// TIA Portal V19 export
FUNCTION_BLOCK "A0302_Centratori_FB"   // FB92, LAD
TITLE = <<< GESTIONE CENTRATORI >>>
// stored: MemoryReserve 100, SetENOAutomatically false
   VAR_INPUT
      AreaInterface : "AreaInterface";
      ZSI : "udt_ZoneSafetyInterface";
      DSI : "udt_DeviceSafetyInterface";
      DataIn : Struct
         OP : "OP_PB";
      END_STRUCT;
      CIn : Struct
         Manager : Struct
            Sollevamento : "ValveMachine_Manager";
            Centraggio : "ValveMachine_Manager";
         END_STRUCT;
         SemiAut_Pb : Bool;
         Rulliera : Struct
            Coda : Struct
               Sens : Struct
                  FTC_Rall : Bool;   // Sensori presenza materiale banco rallentamento ingresso
                  FTC_Prox_Ing : Bool;   // Sensori presenza materiale banco limite ingresso
               END_STRUCT;
            END_STRUCT;
            Centro : Struct
               Sens : Struct
                  FTC_Centrale : Bool;   // 2010BF1 - I50.2
               END_STRUCT;
            END_STRUCT;
         END_STRUCT;
         CarroPareggCoda : Struct
            Ax : "Positioning_DOL_Machine_COut";
            Bloccaggio : "ValveMachine_COut";
            BattutaVerticale : "ValveMachine_COut";
            PareggiatoreLong : "ValveMachine_COut";
            Sens : Struct
               FTC_Ingombro_In : Bool;   // 2012BF1 - I50.0
               FTC_Ingombro_Out : Bool;   // 2012BF2 - I50.1
               PresenzaMat : Bool;   // FC presenza materiale agganciato lato paregg coda
            END_STRUCT;
         END_STRUCT;
         CarroPareggTesta : Struct
            Ax : "Positioning_DOL_Machine_COut";
            Bloccaggio : "ValveMachine_COut";
            Centraggio : "ValveMachine_COut";
            Sollevatore : "ValveMachine_COut";
            Sens : Struct
               FTC1_Rall : Bool;   // 2010BF2 - I50.3
               FTC2_Prox_Ls : Bool;   // 2010BF3 - I50.4
               PresenzaMat : Bool;   // FC presenza materiale agganciato lato paregg testa
            END_STRUCT;
         END_STRUCT;
         BTrk : Struct
            ZoneA0302Entry_Empty : Bool;
            ZoneA0302Exit_Empty : Bool;
         END_STRUCT;
      END_STRUCT;
      Config : Struct
         Centraggio : Array[1..3] of "ValveMachine_Config";
         Sollevamento : Array[1..3] of "ValveMachine_Config";
         DelayMissingCondition : Time;
         WorkWindows : Struct   // Finestre di disattivazione Centratore 1 e 3 in funzione dei Carri
            Coda : Struct
               Min : LReal;
               Max : LReal;
            END_STRUCT;
            Testa : Struct
               Min : LReal;
               Max : LReal;
            END_STRUCT;
         END_STRUCT;
      END_STRUCT;
   END_VAR
   VAR_OUTPUT
      MachineInterface : "MachineInterface";
      COut : Struct
         Centratori : "ValveMachine_COut";
         Centraggio : "ValveMachine_COut";
         Sollevamento : "ValveMachine_COut";
      END_STRUCT;
   END_VAR
   VAR
      Alarm : Struct
         Centraggio : Array[1..3] of "ValveAlr";
         Sollevamento : Array[1..3] of "ValveAlr";
      END_STRUCT;
      Warning : Struct
         Centratore : Array[1..3] of "ValveMachine_Wng";
         Sollevamento : Array[1..3] of "ValveMachine_Wng";
         OP_REST_Centr_MissingCnd : Bool;   // Mancanza comando arresto
         OP_WORK_Centr_MissingCnd : Bool;   // Mancanza consenso lavoro
         OP_REST_Sollev_MissingCnd : Bool;   // Mancanza comando arresto
         OP_WORK_Sollev_MissingCnd : Bool;   // Mancanza consenso lavoro
      END_STRUCT;
      HMI : Struct
         Selection : Struct   // 0=Disable / 1=Enable Pin
            Centraggio : Array[1..3] of Bool;
            Sollevamento : Array[1..3] of Bool;
         END_STRUCT;
         Centratori_Sts : "UDT_HMI-Sts_ValvePosA0301";
         Centraggio_Sts { S7_SetPoint := 'True'} : "UDT_HMI-Sts_ValvePosA0301";
         Sollevamento_Sts { S7_SetPoint := 'True'} : "UDT_HMI-Sts_ValvePosA0301";
      END_STRUCT;
      Centraggio : Array[1..3] of "ValveMachine_FB";
      Sollevamento { S7_SetPoint := 'True'} : Array[1..3] of "ValveMachine_FB";
      Sts : Struct
         Centraggio : Struct
            OP_Rest_Cnd : Bool;
            Op_Work_Cnd : Bool;
         END_STRUCT;
         Sollevamento : Struct
            OP_Rest_Cnd : Bool;
            Op_Work_Cnd : Bool;
         END_STRUCT;
         Centratori_Alarm : Bool;
         Centraggio_AlarmPresence : Bool;
         Sollevamento_AlarmPresence : Bool;
         OP_CanMoveFreely : Bool;
      END_STRUCT;
      Ctrl : Struct
         Centraggio : Struct
            OP_Rest_Man : Bool;
            OP_Work_Man : Bool;
            OP_Rest_Aut : Bool;
            OP_Work_Aut : Bool;
            OP_Rest : Bool;
            OP_Work : Bool;
         END_STRUCT;
         Sollevamento : Struct
            OP_Rest_Man : Bool;
            OP_Work_Man : Bool;
            OP_Rest_Aut : Bool;
            OP_Work_Aut : Bool;
            OP_Rest : Bool;
            OP_Work : Bool;
         END_STRUCT;
      END_STRUCT;
      AUX : Struct
         Centraggio : Struct
            OP_Rest_PB : Bool;
            OP_Work_PB : Bool;
         END_STRUCT;
         Sollevamento : Struct
            OP_Rest_PB : Bool;
            OP_Work_PB : Bool;
         END_STRUCT;
      END_STRUCT;
      TON_OP_REST_Centr_MissingCnd { S7_SetPoint := 'True'} : TON_TIME;
      TON_OP_WORK_Centr_MissingCnd { S7_SetPoint := 'True'} : TON_TIME;
      TON_OP_REST_Sollev_MissingCnd { S7_SetPoint := 'True'} : TON_TIME;
      TON_OP_WORK_Sollev_MissingCnd { S7_SetPoint := 'True'} : TON_TIME;
      DelayMissingCondition : Time;
      TON_Anticipi : Struct
         Work : Struct
            Sollevamento : Array[1..3] of IEC_TIMER;
            Centraggio : Array[1..3] of IEC_TIMER;
         END_STRUCT;
         Rest : Struct
            Sollevamento : Array[1..3] of IEC_TIMER;
            Centraggio : Array[1..3] of IEC_TIMER;
         END_STRUCT;
      END_STRUCT;
   END_VAR
   VAR_TEMP
      PE : Struct
         Centraggio : Struct
            OP_Rest_PB : Bool;
            OP_Work_PB : Bool;
         END_STRUCT;
         Sollevamento : Struct
            OP_Rest_PB : Bool;
            OP_Work_PB : Bool;
         END_STRUCT;
      END_STRUCT;
   END_VAR
   // // Centraggio[1] : Centraggio 1 Coda
   // // Centraggio[2] : Centraggio 2 Centrale
   // // Centraggio[3] : Centraggio 3 Testa
   VAR_TEMP   // added for the SCL form of the ladder/FBD networks
      _w1 : Bool;
      _w2 : Bool;
      _w3 : Bool;
   END_VAR
BEGIN

REGION Network 1: Anticipi Movimento LAVORO
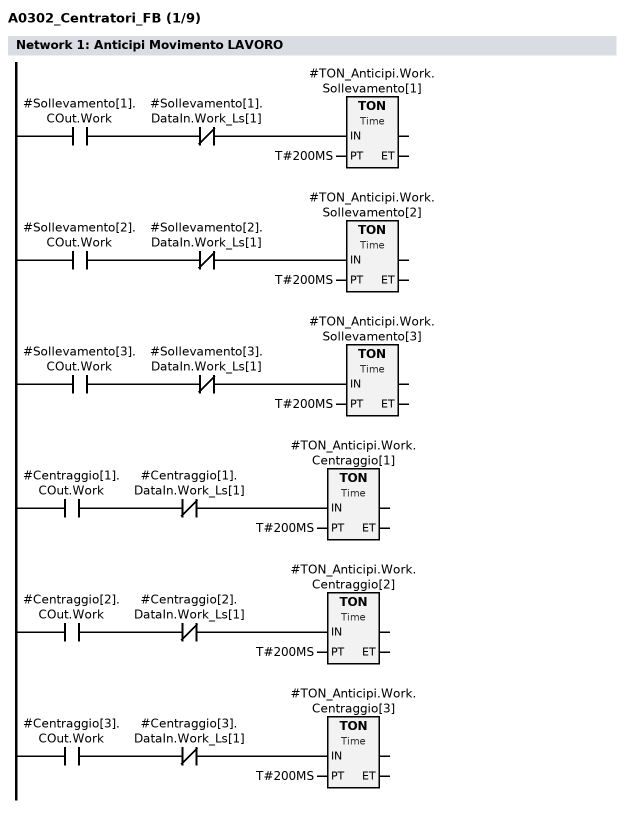
   RUNG wire#powerrail
      Contact( #Sollevamento[1].COut.Work )
      I_Contact( #Sollevamento[1].DataIn.Work_Ls[1] )
      { S7_Templates := "time_type := Time" } #TON_Anticipi.Work.Sollevamento[1].TON(pt := T#200MS, et =>)
   END_RUNG
   RUNG wire#powerrail
      Contact( #Sollevamento[2].COut.Work )
      I_Contact( #Sollevamento[2].DataIn.Work_Ls[1] )
      { S7_Templates := "time_type := Time" } #TON_Anticipi.Work.Sollevamento[2].TON(pt := T#200MS, et =>)
   END_RUNG
   RUNG wire#powerrail
      Contact( #Sollevamento[3].COut.Work )
      I_Contact( #Sollevamento[3].DataIn.Work_Ls[1] )
      { S7_Templates := "time_type := Time" } #TON_Anticipi.Work.Sollevamento[3].TON(pt := T#200MS, et =>)
   END_RUNG
   RUNG wire#powerrail
      Contact( #Centraggio[1].COut.Work )
      I_Contact( #Centraggio[1].DataIn.Work_Ls[1] )
      { S7_Templates := "time_type := Time" } #TON_Anticipi.Work.Centraggio[1].TON(pt := T#200MS, et =>)
   END_RUNG
   RUNG wire#powerrail
      Contact( #Centraggio[2].COut.Work )
      I_Contact( #Centraggio[2].DataIn.Work_Ls[1] )
      { S7_Templates := "time_type := Time" } #TON_Anticipi.Work.Centraggio[2].TON(pt := T#200MS, et =>)
   END_RUNG
   RUNG wire#powerrail
      Contact( #Centraggio[3].COut.Work )
      I_Contact( #Centraggio[3].DataIn.Work_Ls[1] )
      { S7_Templates := "time_type := Time" } #TON_Anticipi.Work.Centraggio[3].TON(pt := T#200MS, et =>)
   END_RUNG
   // the same network as SCL:
   #TON_Anticipi.Work.Sollevamento[1].TON(IN := #Sollevamento[1].COut.Work AND NOT #Sollevamento[1].DataIn.Work_Ls[1],
                           PT := T#200MS);
   #TON_Anticipi.Work.Sollevamento[2].TON(IN := #Sollevamento[2].COut.Work AND NOT #Sollevamento[2].DataIn.Work_Ls[1],
                           PT := T#200MS);
   #TON_Anticipi.Work.Sollevamento[3].TON(IN := #Sollevamento[3].COut.Work AND NOT #Sollevamento[3].DataIn.Work_Ls[1],
                           PT := T#200MS);
   #TON_Anticipi.Work.Centraggio[1].TON(IN := #Centraggio[1].COut.Work AND NOT #Centraggio[1].DataIn.Work_Ls[1],
                           PT := T#200MS);
   #TON_Anticipi.Work.Centraggio[2].TON(IN := #Centraggio[2].COut.Work AND NOT #Centraggio[2].DataIn.Work_Ls[1],
                           PT := T#200MS);
   #TON_Anticipi.Work.Centraggio[3].TON(IN := #Centraggio[3].COut.Work AND NOT #Centraggio[3].DataIn.Work_Ls[1],
                           PT := T#200MS);
END_REGION

REGION Network 2: Anticipi Movimento RIPOSO
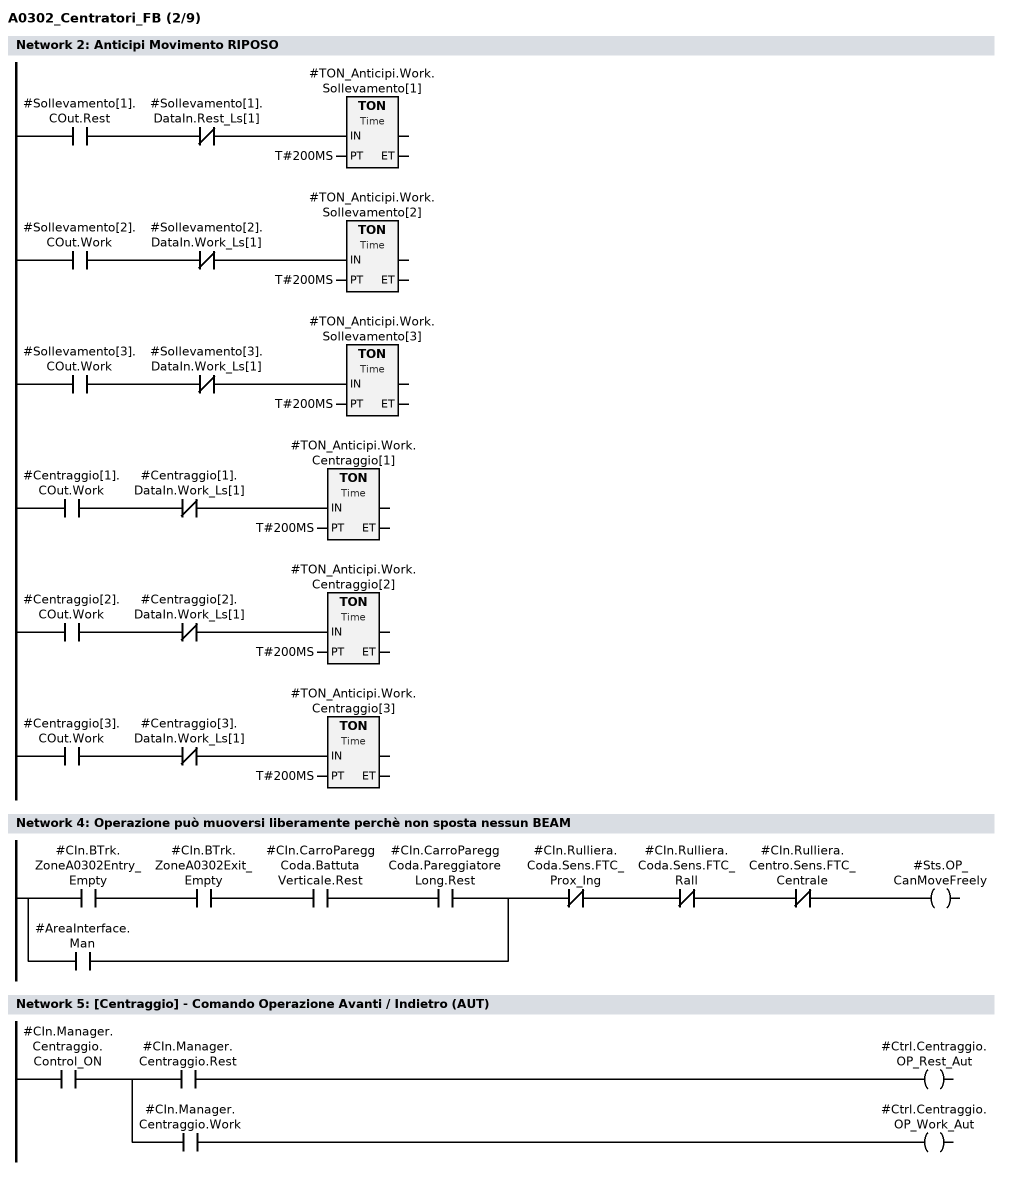
   RUNG wire#powerrail
      Contact( #Sollevamento[1].COut.Rest )
      I_Contact( #Sollevamento[1].DataIn.Rest_Ls[1] )
      { S7_Templates := "time_type := Time" } #TON_Anticipi.Work.Sollevamento[1].TON(pt := T#200MS, et =>)
   END_RUNG
   RUNG wire#powerrail
      Contact( #Sollevamento[2].COut.Work )
      I_Contact( #Sollevamento[2].DataIn.Work_Ls[1] )
      { S7_Templates := "time_type := Time" } #TON_Anticipi.Work.Sollevamento[2].TON(pt := T#200MS, et =>)
   END_RUNG
   RUNG wire#powerrail
      Contact( #Sollevamento[3].COut.Work )
      I_Contact( #Sollevamento[3].DataIn.Work_Ls[1] )
      { S7_Templates := "time_type := Time" } #TON_Anticipi.Work.Sollevamento[3].TON(pt := T#200MS, et =>)
   END_RUNG
   RUNG wire#powerrail
      Contact( #Centraggio[1].COut.Work )
      I_Contact( #Centraggio[1].DataIn.Work_Ls[1] )
      { S7_Templates := "time_type := Time" } #TON_Anticipi.Work.Centraggio[1].TON(pt := T#200MS, et =>)
   END_RUNG
   RUNG wire#powerrail
      Contact( #Centraggio[2].COut.Work )
      I_Contact( #Centraggio[2].DataIn.Work_Ls[1] )
      { S7_Templates := "time_type := Time" } #TON_Anticipi.Work.Centraggio[2].TON(pt := T#200MS, et =>)
   END_RUNG
   RUNG wire#powerrail
      Contact( #Centraggio[3].COut.Work )
      I_Contact( #Centraggio[3].DataIn.Work_Ls[1] )
      { S7_Templates := "time_type := Time" } #TON_Anticipi.Work.Centraggio[3].TON(pt := T#200MS, et =>)
   END_RUNG
   // the same network as SCL:
   #TON_Anticipi.Work.Sollevamento[1].TON(IN := #Sollevamento[1].COut.Rest AND NOT #Sollevamento[1].DataIn.Rest_Ls[1],
                           PT := T#200MS);
   #TON_Anticipi.Work.Sollevamento[2].TON(IN := #Sollevamento[2].COut.Work AND NOT #Sollevamento[2].DataIn.Work_Ls[1],
                           PT := T#200MS);
   #TON_Anticipi.Work.Sollevamento[3].TON(IN := #Sollevamento[3].COut.Work AND NOT #Sollevamento[3].DataIn.Work_Ls[1],
                           PT := T#200MS);
   #TON_Anticipi.Work.Centraggio[1].TON(IN := #Centraggio[1].COut.Work AND NOT #Centraggio[1].DataIn.Work_Ls[1],
                           PT := T#200MS);
   #TON_Anticipi.Work.Centraggio[2].TON(IN := #Centraggio[2].COut.Work AND NOT #Centraggio[2].DataIn.Work_Ls[1],
                           PT := T#200MS);
   #TON_Anticipi.Work.Centraggio[3].TON(IN := #Centraggio[3].COut.Work AND NOT #Centraggio[3].DataIn.Work_Ls[1],
                           PT := T#200MS);
END_REGION

REGION Network 3: <+>
END_REGION

REGION Network 4: Operazione può muoversi liberamente perchè non sposta nessun BEAM
   RUNG wire#powerrail
      Contact( #CIn.BTrk.ZoneA0302Entry_Empty )
      Contact( #CIn.BTrk.ZoneA0302Exit_Empty )
      Contact( #CIn.CarroPareggCoda.BattutaVerticale.Rest )
      Contact( #CIn.CarroPareggCoda.PareggiatoreLong.Rest )
      wire#w1
      I_Contact( #CIn.Rulliera.Coda.Sens.FTC_Prox_Ing )
      I_Contact( #CIn.Rulliera.Coda.Sens.FTC_Rall )
      I_Contact( #CIn.Rulliera.Centro.Sens.FTC_Centrale )
      Coil( #Sts.OP_CanMoveFreely )
   END_RUNG
   RUNG wire#powerrail
      Contact( #AreaInterface.Man )
   END_RUNG wire#w1
   // the same network as SCL:
   #Sts.OP_CanMoveFreely := ((#CIn.BTrk.ZoneA0302Entry_Empty AND #CIn.BTrk.ZoneA0302Exit_Empty AND #CIn.CarroPareggCoda.BattutaVerticale.Rest AND #CIn.CarroPareggCoda.PareggiatoreLong.Rest) OR #AreaInterface.Man) AND NOT #CIn.Rulliera.Coda.Sens.FTC_Prox_Ing AND NOT #CIn.Rulliera.Coda.Sens.FTC_Rall AND NOT #CIn.Rulliera.Centro.Sens.FTC_Centrale;
END_REGION

REGION Network 5: [Centraggio] - Comando Operazione Avanti / Indietro (AUT)
   RUNG wire#powerrail
      Contact( #CIn.Manager.Centraggio.Control_ON )
      wire#w1
      Contact( #CIn.Manager.Centraggio.Rest )
      Coil( #Ctrl.Centraggio.OP_Rest_Aut )
   END_RUNG
   RUNG wire#w1
      Contact( #CIn.Manager.Centraggio.Work )
      Coil( #Ctrl.Centraggio.OP_Work_Aut )
   END_RUNG
   // the same network as SCL:
   #Ctrl.Centraggio.OP_Rest_Aut := #CIn.Manager.Centraggio.Control_ON AND #CIn.Manager.Centraggio.Rest;
   #Ctrl.Centraggio.OP_Work_Aut := #CIn.Manager.Centraggio.Control_ON AND #CIn.Manager.Centraggio.Work;
END_REGION

REGION Network 6: [Centraggio] - Comando Operazione Lavoro / Riposo (MAN)
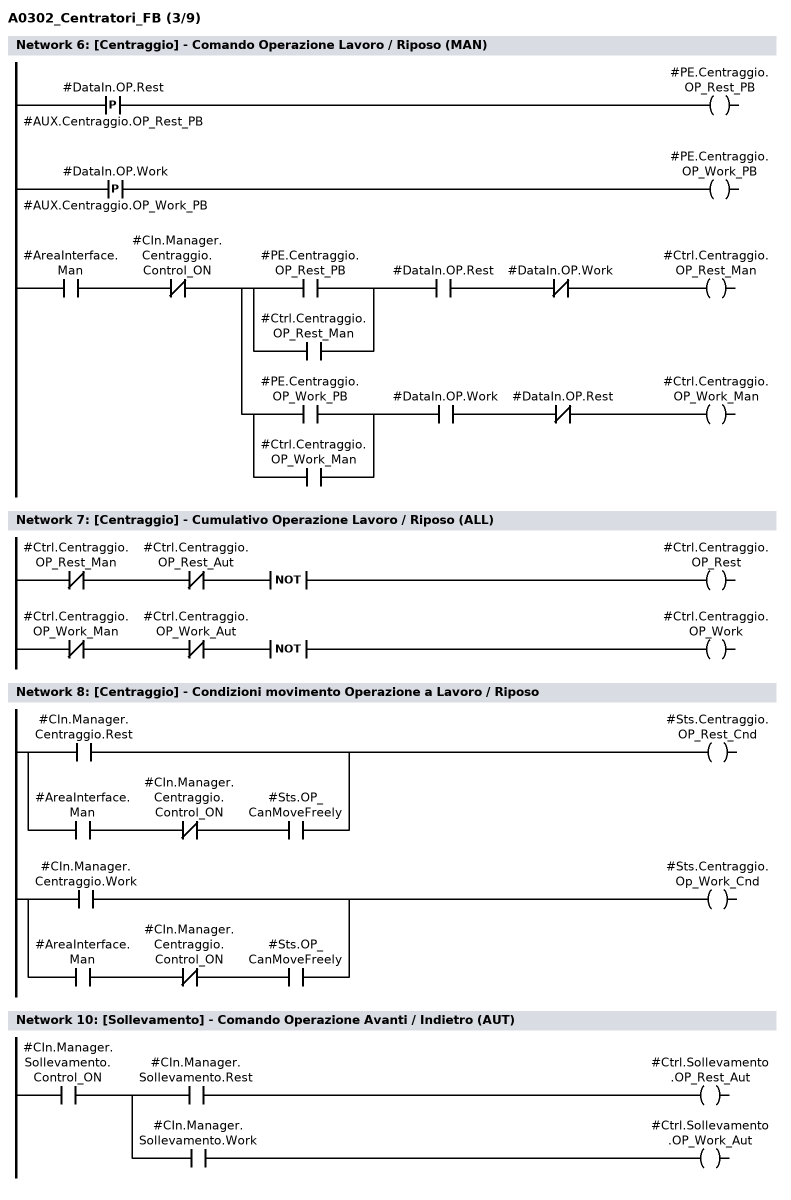
   RUNG wire#powerrail
      P_Contact(operand := #DataIn.OP.Rest, bit := #AUX.Centraggio.OP_Rest_PB)
      Coil( #PE.Centraggio.OP_Rest_PB )
   END_RUNG
   RUNG wire#powerrail
      P_Contact(operand := #DataIn.OP.Work, bit := #AUX.Centraggio.OP_Work_PB)
      Coil( #PE.Centraggio.OP_Work_PB )
   END_RUNG
   RUNG wire#powerrail
      Contact( #AreaInterface.Man )
      I_Contact( #CIn.Manager.Centraggio.Control_ON )
      wire#w1
      Contact( #PE.Centraggio.OP_Rest_PB )
      wire#w2
      Contact( #DataIn.OP.Rest )
      I_Contact( #DataIn.OP.Work )
      Coil( #Ctrl.Centraggio.OP_Rest_Man )
   END_RUNG
   RUNG wire#w1
      Contact( #Ctrl.Centraggio.OP_Rest_Man )
   END_RUNG wire#w2
   RUNG wire#w1
      Contact( #PE.Centraggio.OP_Work_PB )
      wire#w3
      Contact( #DataIn.OP.Work )
      I_Contact( #DataIn.OP.Rest )
      Coil( #Ctrl.Centraggio.OP_Work_Man )
   END_RUNG
   RUNG wire#w1
      Contact( #Ctrl.Centraggio.OP_Work_Man )
   END_RUNG wire#w3
   // the same network as SCL:
   #_w1 := #DataIn.OP.Rest AND NOT #AUX.Centraggio.OP_Rest_PB;   // rising edge of #DataIn.OP.Rest
   #AUX.Centraggio.OP_Rest_PB := #DataIn.OP.Rest;
   #PE.Centraggio.OP_Rest_PB := #_w1;
   #_w2 := #DataIn.OP.Work AND NOT #AUX.Centraggio.OP_Work_PB;   // rising edge of #DataIn.OP.Work
   #AUX.Centraggio.OP_Work_PB := #DataIn.OP.Work;
   #PE.Centraggio.OP_Work_PB := #_w2;
   #_w3 := #AreaInterface.Man AND NOT #CIn.Manager.Centraggio.Control_ON;
   #Ctrl.Centraggio.OP_Rest_Man := #_w3 AND (#PE.Centraggio.OP_Rest_PB OR #Ctrl.Centraggio.OP_Rest_Man) AND #DataIn.OP.Rest AND NOT #DataIn.OP.Work;
   #Ctrl.Centraggio.OP_Work_Man := #_w3 AND (#PE.Centraggio.OP_Work_PB OR #Ctrl.Centraggio.OP_Work_Man) AND #DataIn.OP.Work AND NOT #DataIn.OP.Rest;
END_REGION

REGION Network 7: [Centraggio] - Cumulativo Operazione Lavoro / Riposo (ALL)
   RUNG wire#powerrail
      I_Contact( #Ctrl.Centraggio.OP_Rest_Man )
      I_Contact( #Ctrl.Centraggio.OP_Rest_Aut )
      Not()
      Coil( #Ctrl.Centraggio.OP_Rest )
   END_RUNG
   RUNG wire#powerrail
      I_Contact( #Ctrl.Centraggio.OP_Work_Man )
      I_Contact( #Ctrl.Centraggio.OP_Work_Aut )
      Not()
      Coil( #Ctrl.Centraggio.OP_Work )
   END_RUNG
   // the same network as SCL:
   #Ctrl.Centraggio.OP_Rest := NOT (NOT #Ctrl.Centraggio.OP_Rest_Man AND NOT #Ctrl.Centraggio.OP_Rest_Aut);
   #Ctrl.Centraggio.OP_Work := NOT (NOT #Ctrl.Centraggio.OP_Work_Man AND NOT #Ctrl.Centraggio.OP_Work_Aut);
END_REGION

REGION Network 8: [Centraggio] - Condizioni movimento Operazione a Lavoro / Riposo
   RUNG wire#powerrail
      Contact( #CIn.Manager.Centraggio.Rest )
      wire#w1
      Coil( #Sts.Centraggio.OP_Rest_Cnd )
   END_RUNG
   RUNG wire#powerrail
      Contact( #AreaInterface.Man )
      I_Contact( #CIn.Manager.Centraggio.Control_ON )
      Contact( #Sts.OP_CanMoveFreely )
   END_RUNG wire#w1
   RUNG wire#powerrail
      Contact( #CIn.Manager.Centraggio.Work )
      wire#w2
      Coil( #Sts.Centraggio.Op_Work_Cnd )
   END_RUNG
   RUNG wire#powerrail
      Contact( #AreaInterface.Man )
      I_Contact( #CIn.Manager.Centraggio.Control_ON )
      Contact( #Sts.OP_CanMoveFreely )
   END_RUNG wire#w2
   // the same network as SCL:
   #Sts.Centraggio.OP_Rest_Cnd := #CIn.Manager.Centraggio.Rest OR (#AreaInterface.Man AND NOT #CIn.Manager.Centraggio.Control_ON AND #Sts.OP_CanMoveFreely);
   #Sts.Centraggio.Op_Work_Cnd := #CIn.Manager.Centraggio.Work OR (#AreaInterface.Man AND NOT #CIn.Manager.Centraggio.Control_ON AND #Sts.OP_CanMoveFreely);
END_REGION

REGION Network 10: [Sollevamento] - Comando Operazione Avanti / Indietro (AUT)
   RUNG wire#powerrail
      Contact( #CIn.Manager.Sollevamento.Control_ON )
      wire#w1
      Contact( #CIn.Manager.Sollevamento.Rest )
      Coil( #Ctrl.Sollevamento.OP_Rest_Aut )
   END_RUNG
   RUNG wire#w1
      Contact( #CIn.Manager.Sollevamento.Work )
      Coil( #Ctrl.Sollevamento.OP_Work_Aut )
   END_RUNG
   // the same network as SCL:
   #Ctrl.Sollevamento.OP_Rest_Aut := #CIn.Manager.Sollevamento.Control_ON AND #CIn.Manager.Sollevamento.Rest;
   #Ctrl.Sollevamento.OP_Work_Aut := #CIn.Manager.Sollevamento.Control_ON AND #CIn.Manager.Sollevamento.Work;
END_REGION

REGION Network 11: [Sollevamento] - Comando Operazione Lavoro / Riposo (MAN)
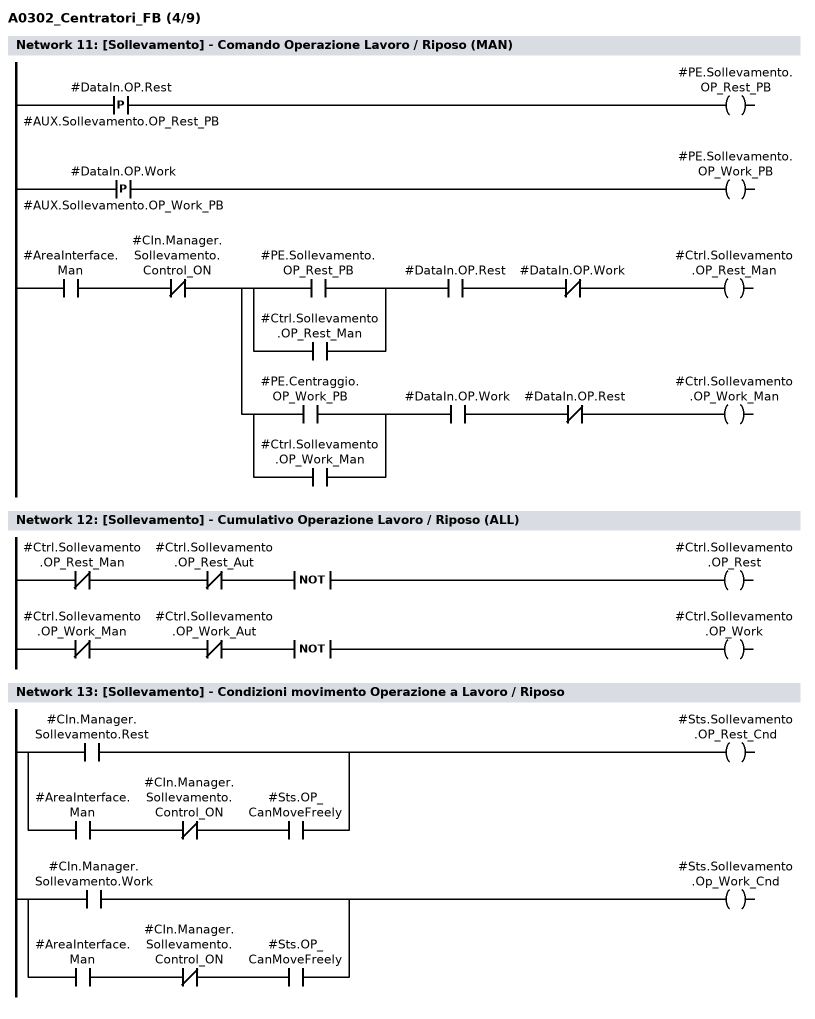
   RUNG wire#powerrail
      P_Contact(operand := #DataIn.OP.Rest, bit := #AUX.Sollevamento.OP_Rest_PB)
      Coil( #PE.Sollevamento.OP_Rest_PB )
   END_RUNG
   RUNG wire#powerrail
      P_Contact(operand := #DataIn.OP.Work, bit := #AUX.Sollevamento.OP_Work_PB)
      Coil( #PE.Sollevamento.OP_Work_PB )
   END_RUNG
   RUNG wire#powerrail
      Contact( #AreaInterface.Man )
      I_Contact( #CIn.Manager.Sollevamento.Control_ON )
      wire#w1
      Contact( #PE.Sollevamento.OP_Rest_PB )
      wire#w2
      Contact( #DataIn.OP.Rest )
      I_Contact( #DataIn.OP.Work )
      Coil( #Ctrl.Sollevamento.OP_Rest_Man )
   END_RUNG
   RUNG wire#w1
      Contact( #Ctrl.Sollevamento.OP_Rest_Man )
   END_RUNG wire#w2
   RUNG wire#w1
      Contact( #PE.Centraggio.OP_Work_PB )
      wire#w3
      Contact( #DataIn.OP.Work )
      I_Contact( #DataIn.OP.Rest )
      Coil( #Ctrl.Sollevamento.OP_Work_Man )
   END_RUNG
   RUNG wire#w1
      Contact( #Ctrl.Sollevamento.OP_Work_Man )
   END_RUNG wire#w3
   // the same network as SCL:
   #_w1 := #DataIn.OP.Rest AND NOT #AUX.Sollevamento.OP_Rest_PB;   // rising edge of #DataIn.OP.Rest
   #AUX.Sollevamento.OP_Rest_PB := #DataIn.OP.Rest;
   #PE.Sollevamento.OP_Rest_PB := #_w1;
   #_w2 := #DataIn.OP.Work AND NOT #AUX.Sollevamento.OP_Work_PB;   // rising edge of #DataIn.OP.Work
   #AUX.Sollevamento.OP_Work_PB := #DataIn.OP.Work;
   #PE.Sollevamento.OP_Work_PB := #_w2;
   #_w3 := #AreaInterface.Man AND NOT #CIn.Manager.Sollevamento.Control_ON;
   #Ctrl.Sollevamento.OP_Rest_Man := #_w3 AND (#PE.Sollevamento.OP_Rest_PB OR #Ctrl.Sollevamento.OP_Rest_Man) AND #DataIn.OP.Rest AND NOT #DataIn.OP.Work;
   #Ctrl.Sollevamento.OP_Work_Man := #_w3 AND (#PE.Centraggio.OP_Work_PB OR #Ctrl.Sollevamento.OP_Work_Man) AND #DataIn.OP.Work AND NOT #DataIn.OP.Rest;
END_REGION

REGION Network 12: [Sollevamento] - Cumulativo Operazione Lavoro / Riposo (ALL)
   RUNG wire#powerrail
      I_Contact( #Ctrl.Sollevamento.OP_Rest_Man )
      I_Contact( #Ctrl.Sollevamento.OP_Rest_Aut )
      Not()
      Coil( #Ctrl.Sollevamento.OP_Rest )
   END_RUNG
   RUNG wire#powerrail
      I_Contact( #Ctrl.Sollevamento.OP_Work_Man )
      I_Contact( #Ctrl.Sollevamento.OP_Work_Aut )
      Not()
      Coil( #Ctrl.Sollevamento.OP_Work )
   END_RUNG
   // the same network as SCL:
   #Ctrl.Sollevamento.OP_Rest := NOT (NOT #Ctrl.Sollevamento.OP_Rest_Man AND NOT #Ctrl.Sollevamento.OP_Rest_Aut);
   #Ctrl.Sollevamento.OP_Work := NOT (NOT #Ctrl.Sollevamento.OP_Work_Man AND NOT #Ctrl.Sollevamento.OP_Work_Aut);
END_REGION

REGION Network 13: [Sollevamento] - Condizioni movimento Operazione a Lavoro / Riposo
   RUNG wire#powerrail
      Contact( #CIn.Manager.Sollevamento.Rest )
      wire#w1
      Coil( #Sts.Sollevamento.OP_Rest_Cnd )
   END_RUNG
   RUNG wire#powerrail
      Contact( #AreaInterface.Man )
      I_Contact( #CIn.Manager.Sollevamento.Control_ON )
      Contact( #Sts.OP_CanMoveFreely )
   END_RUNG wire#w1
   RUNG wire#powerrail
      Contact( #CIn.Manager.Sollevamento.Work )
      wire#w2
      Coil( #Sts.Sollevamento.Op_Work_Cnd )
   END_RUNG
   RUNG wire#powerrail
      Contact( #AreaInterface.Man )
      I_Contact( #CIn.Manager.Sollevamento.Control_ON )
      Contact( #Sts.OP_CanMoveFreely )
   END_RUNG wire#w2
   // the same network as SCL:
   #Sts.Sollevamento.OP_Rest_Cnd := #CIn.Manager.Sollevamento.Rest OR (#AreaInterface.Man AND NOT #CIn.Manager.Sollevamento.Control_ON AND #Sts.OP_CanMoveFreely);
   #Sts.Sollevamento.Op_Work_Cnd := #CIn.Manager.Sollevamento.Work OR (#AreaInterface.Man AND NOT #CIn.Manager.Sollevamento.Control_ON AND #Sts.OP_CanMoveFreely);
END_REGION

REGION Network 15 (SCL): Centraggio + Sollevamento - Cin Manager (Esecuzione sequenza comandi)
   //
   #Centraggio[1].Cin.Manager.Control_ON := #Centraggio[2].Cin.Manager.Control_ON :=
   #Centraggio[3].Cin.Manager.Control_ON := #CIn.Manager.Centraggio.Control_ON;
   //
   #Sollevamento[1].Cin.Manager.Control_ON :=#Sollevamento[2].Cin.Manager.Control_ON :=
   #Sollevamento[3].Cin.Manager.Control_ON := #CIn.Manager.Sollevamento.Control_ON;

   REGION Se nessun comando attivo resetto il comando Work/Rest
       #Centraggio[1].Cin.Manager.Rest := FALSE;
       #Centraggio[2].Cin.Manager.Rest := FALSE;
       #Centraggio[3].Cin.Manager.Rest := FALSE;

       #Centraggio[1].Cin.Manager.Work := FALSE;
       #Centraggio[2].Cin.Manager.Work := FALSE;
       #Centraggio[3].Cin.Manager.Work := FALSE;

       #Sollevamento[1].Cin.Manager.Rest := FALSE;
       #Sollevamento[2].Cin.Manager.Rest := FALSE;
       #Sollevamento[3].Cin.Manager.Rest := FALSE;

       #Sollevamento[1].Cin.Manager.Work := FALSE;
       #Sollevamento[2].Cin.Manager.Work := FALSE;
       #Sollevamento[3].Cin.Manager.Work := FALSE;
   END_REGION ;


   IF #AreaInterface.Aut OR #CIn.SemiAut_Pb THEN

       IF #Ctrl.Sollevamento.OP_Rest AND #Sts.Sollevamento.OP_Rest_Cnd
           AND #Centraggio[2].COut.Rest THEN
           #Sollevamento[1].Cin.Manager.Rest := TRUE;
           #Sollevamento[2].Cin.Manager.Rest := TRUE;
           #Sollevamento[3].Cin.Manager.Rest := TRUE;

       ELSIF #Ctrl.Sollevamento.OP_Work AND #Sts.Sollevamento.Op_Work_Cnd THEN
           #Sollevamento[1].Cin.Manager.Work := TRUE;
           #Sollevamento[2].Cin.Manager.Work := TRUE;
           #Sollevamento[3].Cin.Manager.Work := TRUE;

       END_IF;


       IF #Ctrl.Centraggio.OP_Rest AND #Sts.Centraggio.OP_Rest_Cnd THEN
           #Centraggio[1].Cin.Manager.Rest := TRUE;
           #Centraggio[2].Cin.Manager.Rest := TRUE;
           #Centraggio[3].Cin.Manager.Rest := TRUE;

       ELSIF #Ctrl.Centraggio.OP_Work AND #Sts.Centraggio.Op_Work_Cnd
           AND #Sollevamento[2].COut.Work THEN
           #Centraggio[1].Cin.Manager.Work := TRUE;
           #Centraggio[2].Cin.Manager.Work := TRUE;
           #Centraggio[3].Cin.Manager.Work := TRUE;

       END_IF;
   END_IF;
END_REGION

REGION Network 16 (SCL): Centraggio + Sollevamento - CIn Abilitazioni Manager
   #Centraggio[1].Cin.Manager.EnableStopDoorOpeningReq := #Centraggio[2].Cin.Manager.EnableStopDoorOpeningReq :=
   #Centraggio[3].Cin.Manager.EnableStopDoorOpeningReq := #CIn.Manager.Centraggio.EnableStopDoorOpeningReq;

   #Sollevamento[1].Cin.Manager.EnableStopDoorOpeningReq := #Sollevamento[2].Cin.Manager.EnableStopDoorOpeningReq :=
   #Sollevamento[3].Cin.Manager.EnableStopDoorOpeningReq := #CIn.Manager.Sollevamento.EnableStopDoorOpeningReq;

   #Centraggio[1].Cin.Manager.EnableStopInPhase := #Centraggio[2].Cin.Manager.EnableStopInPhase :=
   #Centraggio[3].Cin.Manager.EnableStopInPhase := #CIn.Manager.Centraggio.EnableStopInPhase;

   #Sollevamento[1].Cin.Manager.EnableStopInPhase :=#Sollevamento[2].Cin.Manager.EnableStopInPhase:=
   #Sollevamento[3].Cin.Manager.EnableStopInPhase:= #CIn.Manager.Sollevamento.EnableStopInPhase;

   #Centraggio[1].Cin.Manager.EnableStopProgrammed := #Centraggio[2].Cin.Manager.EnableStopProgrammed
   := #Centraggio[3].Cin.Manager.EnableStopProgrammed := #CIn.Manager.Centraggio.EnableStopProgrammed;

   #Sollevamento[1].Cin.Manager.EnableStopProgrammed :=#Sollevamento[2].Cin.Manager.EnableStopProgrammed:=
   #Sollevamento[3].Cin.Manager.EnableStopProgrammed:=  #CIn.Manager.Sollevamento.EnableStopProgrammed;
END_REGION

REGION Network 17: <+>
END_REGION

REGION Network 18: [Centraggio] - Warning manacanza condizioni esecuzione Operazione RIPOSO / LAVORO
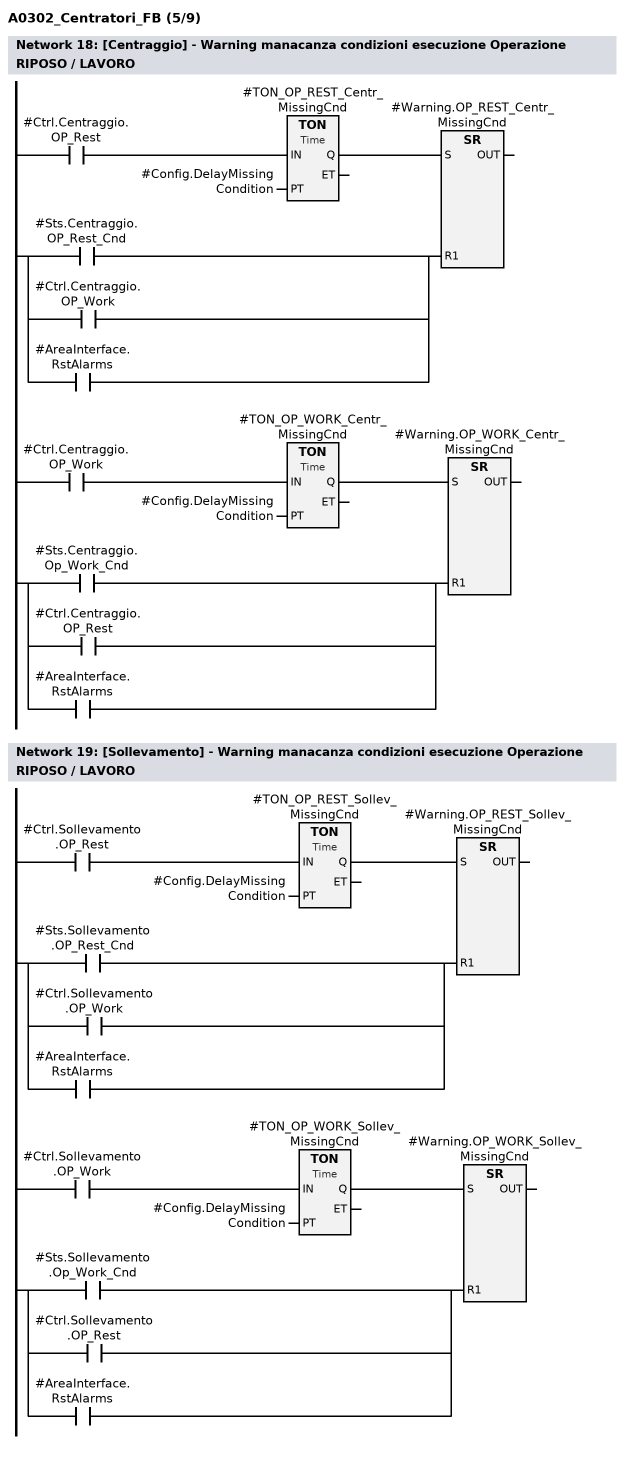
   RUNG wire#powerrail
      Contact( #Ctrl.Centraggio.OP_Rest )
      { S7_Templates := "time_type := Time" } #TON_OP_REST_Centr_MissingCnd.TON(pt := #Config.DelayMissingCondition, et =>)
      S_SR(operand := #Warning.OP_REST_Centr_MissingCnd, r1 := wire#w1)
   END_RUNG
   RUNG wire#powerrail
      Contact( #Sts.Centraggio.OP_Rest_Cnd )
   END_RUNG wire#w1
   RUNG wire#powerrail
      Contact( #Ctrl.Centraggio.OP_Work )
   END_RUNG wire#w1
   RUNG wire#powerrail
      Contact( #AreaInterface.RstAlarms )
   END_RUNG wire#w1
   RUNG wire#powerrail
      Contact( #Ctrl.Centraggio.OP_Work )
      { S7_Templates := "time_type := Time" } #TON_OP_WORK_Centr_MissingCnd.TON(pt := #Config.DelayMissingCondition, et =>)
      S_SR(operand := #Warning.OP_WORK_Centr_MissingCnd, r1 := wire#w2)
   END_RUNG
   RUNG wire#powerrail
      Contact( #Sts.Centraggio.Op_Work_Cnd )
   END_RUNG wire#w2
   RUNG wire#powerrail
      Contact( #Ctrl.Centraggio.OP_Rest )
   END_RUNG wire#w2
   RUNG wire#powerrail
      Contact( #AreaInterface.RstAlarms )
   END_RUNG wire#w2
   // the same network as SCL:
   #TON_OP_REST_Centr_MissingCnd(IN := #Ctrl.Centraggio.OP_Rest, PT := #Config.DelayMissingCondition);   // TON
   IF #TON_OP_REST_Centr_MissingCnd.Q THEN
       #Warning.OP_REST_Centr_MissingCnd := TRUE;   // SR flip-flop
   END_IF;
   IF #Sts.Centraggio.OP_Rest_Cnd OR #Ctrl.Centraggio.OP_Work OR #AreaInterface.RstAlarms THEN
       #Warning.OP_REST_Centr_MissingCnd := FALSE;
   END_IF;
   #TON_OP_WORK_Centr_MissingCnd(IN := #Ctrl.Centraggio.OP_Work, PT := #Config.DelayMissingCondition);   // TON
   IF #TON_OP_WORK_Centr_MissingCnd.Q THEN
       #Warning.OP_WORK_Centr_MissingCnd := TRUE;   // SR flip-flop
   END_IF;
   IF #Sts.Centraggio.Op_Work_Cnd OR #Ctrl.Centraggio.OP_Rest OR #AreaInterface.RstAlarms THEN
       #Warning.OP_WORK_Centr_MissingCnd := FALSE;
   END_IF;
END_REGION

REGION Network 19: [Sollevamento] - Warning manacanza condizioni esecuzione Operazione RIPOSO / LAVORO
   RUNG wire#powerrail
      Contact( #Ctrl.Sollevamento.OP_Rest )
      { S7_Templates := "time_type := Time" } #TON_OP_REST_Sollev_MissingCnd.TON(pt := #Config.DelayMissingCondition, et =>)
      S_SR(operand := #Warning.OP_REST_Sollev_MissingCnd, r1 := wire#w1)
   END_RUNG
   RUNG wire#powerrail
      Contact( #Sts.Sollevamento.OP_Rest_Cnd )
   END_RUNG wire#w1
   RUNG wire#powerrail
      Contact( #Ctrl.Sollevamento.OP_Work )
   END_RUNG wire#w1
   RUNG wire#powerrail
      Contact( #AreaInterface.RstAlarms )
   END_RUNG wire#w1
   RUNG wire#powerrail
      Contact( #Ctrl.Sollevamento.OP_Work )
      { S7_Templates := "time_type := Time" } #TON_OP_WORK_Sollev_MissingCnd.TON(pt := #Config.DelayMissingCondition, et =>)
      S_SR(operand := #Warning.OP_WORK_Sollev_MissingCnd, r1 := wire#w2)
   END_RUNG
   RUNG wire#powerrail
      Contact( #Sts.Sollevamento.Op_Work_Cnd )
   END_RUNG wire#w2
   RUNG wire#powerrail
      Contact( #Ctrl.Sollevamento.OP_Rest )
   END_RUNG wire#w2
   RUNG wire#powerrail
      Contact( #AreaInterface.RstAlarms )
   END_RUNG wire#w2
   // the same network as SCL:
   #TON_OP_REST_Sollev_MissingCnd(IN := #Ctrl.Sollevamento.OP_Rest, PT := #Config.DelayMissingCondition);   // TON
   IF #TON_OP_REST_Sollev_MissingCnd.Q THEN
       #Warning.OP_REST_Sollev_MissingCnd := TRUE;   // SR flip-flop
   END_IF;
   IF #Sts.Sollevamento.OP_Rest_Cnd OR #Ctrl.Sollevamento.OP_Work OR #AreaInterface.RstAlarms THEN
       #Warning.OP_REST_Sollev_MissingCnd := FALSE;
   END_IF;
   #TON_OP_WORK_Sollev_MissingCnd(IN := #Ctrl.Sollevamento.OP_Work, PT := #Config.DelayMissingCondition);   // TON
   IF #TON_OP_WORK_Sollev_MissingCnd.Q THEN
       #Warning.OP_WORK_Sollev_MissingCnd := TRUE;   // SR flip-flop
   END_IF;
   IF #Sts.Sollevamento.Op_Work_Cnd OR #Ctrl.Sollevamento.OP_Rest OR #AreaInterface.RstAlarms THEN
       #Warning.OP_WORK_Sollev_MissingCnd := FALSE;
   END_IF;
END_REGION

REGION Network 21: Centraggio - CIn External alarm
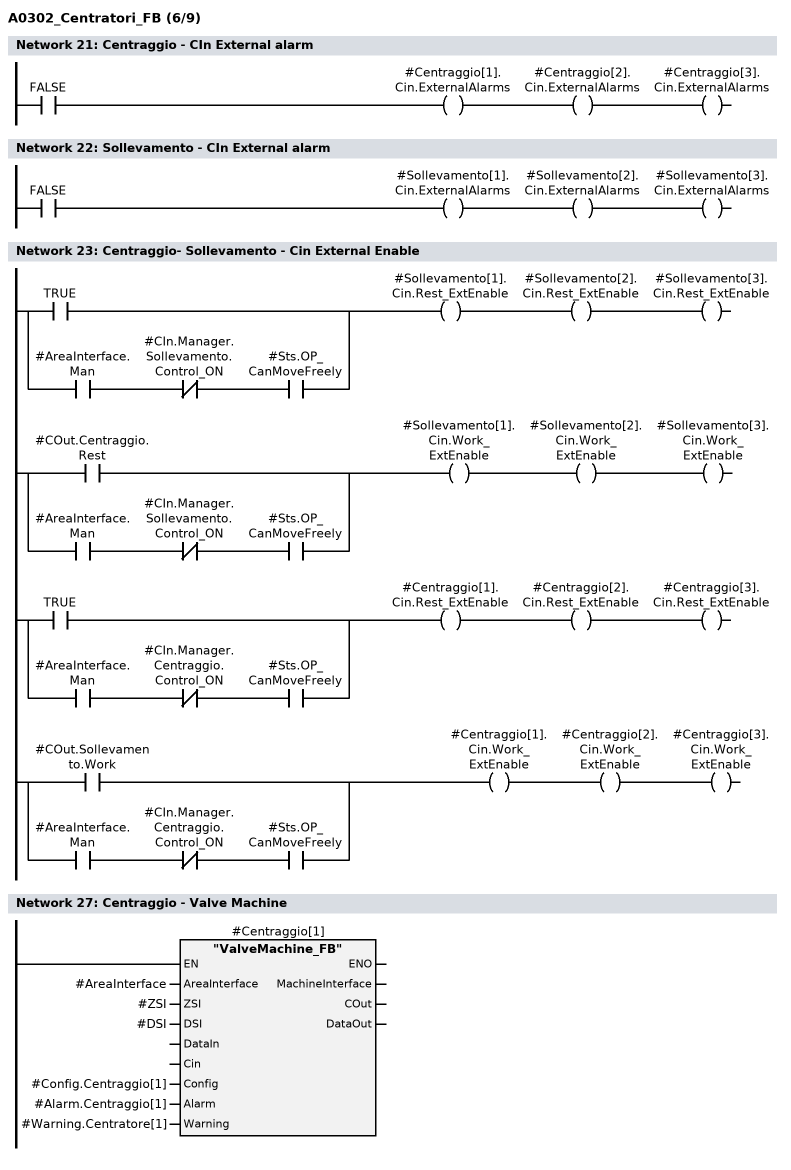
   RUNG wire#powerrail
      Contact( FALSE )
      Coil( #Centraggio[1].Cin.ExternalAlarms )
      Coil( #Centraggio[2].Cin.ExternalAlarms )
      Coil( #Centraggio[3].Cin.ExternalAlarms )
   END_RUNG
   // the same network as SCL:
   #Centraggio[1].Cin.ExternalAlarms := FALSE;
   #Centraggio[2].Cin.ExternalAlarms := FALSE;
   #Centraggio[3].Cin.ExternalAlarms := FALSE;
END_REGION

REGION Network 22: Sollevamento - CIn External alarm
   RUNG wire#powerrail
      Contact( FALSE )
      Coil( #Sollevamento[1].Cin.ExternalAlarms )
      Coil( #Sollevamento[2].Cin.ExternalAlarms )
      Coil( #Sollevamento[3].Cin.ExternalAlarms )
   END_RUNG
   // the same network as SCL:
   #Sollevamento[1].Cin.ExternalAlarms := FALSE;
   #Sollevamento[2].Cin.ExternalAlarms := FALSE;
   #Sollevamento[3].Cin.ExternalAlarms := FALSE;
END_REGION

REGION Network 23: Centraggio- Sollevamento - Cin External Enable
   RUNG wire#powerrail
      Contact( TRUE )
      wire#w1
      Coil( #Sollevamento[1].Cin.Rest_ExtEnable )
      Coil( #Sollevamento[2].Cin.Rest_ExtEnable )
      Coil( #Sollevamento[3].Cin.Rest_ExtEnable )
   END_RUNG
   RUNG wire#powerrail
      Contact( #AreaInterface.Man )
      I_Contact( #CIn.Manager.Sollevamento.Control_ON )
      Contact( #Sts.OP_CanMoveFreely )
   END_RUNG wire#w1
   RUNG wire#powerrail
      Contact( #COut.Centraggio.Rest )
      wire#w2
      Coil( #Sollevamento[1].Cin.Work_ExtEnable )
      Coil( #Sollevamento[2].Cin.Work_ExtEnable )
      Coil( #Sollevamento[3].Cin.Work_ExtEnable )
   END_RUNG
   RUNG wire#powerrail
      Contact( #AreaInterface.Man )
      I_Contact( #CIn.Manager.Sollevamento.Control_ON )
      Contact( #Sts.OP_CanMoveFreely )
   END_RUNG wire#w2
   RUNG wire#powerrail
      Contact( TRUE )
      wire#w3
      Coil( #Centraggio[1].Cin.Rest_ExtEnable )
      Coil( #Centraggio[2].Cin.Rest_ExtEnable )
      Coil( #Centraggio[3].Cin.Rest_ExtEnable )
   END_RUNG
   RUNG wire#powerrail
      Contact( #AreaInterface.Man )
      I_Contact( #CIn.Manager.Centraggio.Control_ON )
      Contact( #Sts.OP_CanMoveFreely )
   END_RUNG wire#w3
   RUNG wire#powerrail
      Contact( #COut.Sollevamento.Work )
      wire#w4
      Coil( #Centraggio[1].Cin.Work_ExtEnable )
      Coil( #Centraggio[2].Cin.Work_ExtEnable )
      Coil( #Centraggio[3].Cin.Work_ExtEnable )
   END_RUNG
   RUNG wire#powerrail
      Contact( #AreaInterface.Man )
      I_Contact( #CIn.Manager.Centraggio.Control_ON )
      Contact( #Sts.OP_CanMoveFreely )
   END_RUNG wire#w4
   // the same network as SCL:
   #Sollevamento[1].Cin.Rest_ExtEnable := TRUE OR (#AreaInterface.Man AND NOT #CIn.Manager.Sollevamento.Control_ON AND #Sts.OP_CanMoveFreely);
   #Sollevamento[2].Cin.Rest_ExtEnable := TRUE OR (#AreaInterface.Man AND NOT #CIn.Manager.Sollevamento.Control_ON AND #Sts.OP_CanMoveFreely);
   #Sollevamento[3].Cin.Rest_ExtEnable := TRUE OR (#AreaInterface.Man AND NOT #CIn.Manager.Sollevamento.Control_ON AND #Sts.OP_CanMoveFreely);
   #Sollevamento[1].Cin.Work_ExtEnable := #COut.Centraggio.Rest OR (#AreaInterface.Man AND NOT #CIn.Manager.Sollevamento.Control_ON AND #Sts.OP_CanMoveFreely);
   #Sollevamento[2].Cin.Work_ExtEnable := #COut.Centraggio.Rest OR (#AreaInterface.Man AND NOT #CIn.Manager.Sollevamento.Control_ON AND #Sts.OP_CanMoveFreely);
   #Sollevamento[3].Cin.Work_ExtEnable := #COut.Centraggio.Rest OR (#AreaInterface.Man AND NOT #CIn.Manager.Sollevamento.Control_ON AND #Sts.OP_CanMoveFreely);
   #Centraggio[1].Cin.Rest_ExtEnable := TRUE OR (#AreaInterface.Man AND NOT #CIn.Manager.Centraggio.Control_ON AND #Sts.OP_CanMoveFreely);
   #Centraggio[2].Cin.Rest_ExtEnable := TRUE OR (#AreaInterface.Man AND NOT #CIn.Manager.Centraggio.Control_ON AND #Sts.OP_CanMoveFreely);
   #Centraggio[3].Cin.Rest_ExtEnable := TRUE OR (#AreaInterface.Man AND NOT #CIn.Manager.Centraggio.Control_ON AND #Sts.OP_CanMoveFreely);
   #Centraggio[1].Cin.Work_ExtEnable := #COut.Sollevamento.Work OR (#AreaInterface.Man AND NOT #CIn.Manager.Centraggio.Control_ON AND #Sts.OP_CanMoveFreely);
   #Centraggio[2].Cin.Work_ExtEnable := #COut.Sollevamento.Work OR (#AreaInterface.Man AND NOT #CIn.Manager.Centraggio.Control_ON AND #Sts.OP_CanMoveFreely);
   #Centraggio[3].Cin.Work_ExtEnable := #COut.Sollevamento.Work OR (#AreaInterface.Man AND NOT #CIn.Manager.Centraggio.Control_ON AND #Sts.OP_CanMoveFreely);
END_REGION

REGION Network 25: <<< CENTRATORE 1 TESTA >>>
END_REGION

REGION Network 26 (SCL): Centraggio - Finestra di lavoro - Enable/Disable
   // Disattivazione Centratore lato Testa in funzione della posizione del Carro Pareggiatore Testa
   // 

   IF #CIn.CarroPareggTesta.Ax.Homed THEN

       IF #CIn.CarroPareggTesta.Ax.ActualPosition >= "PrjConfig_A03".A0302.Centratori.WorkWindows.Testa.Min AND
           #CIn.CarroPareggTesta.Ax.ActualPosition < "PrjConfig_A03".A0302.Centratori.WorkWindows.Testa.Max THEN
           #Sollevamento[1].Cin.Manager.Rest := TRUE;
           #Centraggio[1].Cin.Manager.Rest := TRUE;
           #HMI.Selection.Sollevamento[1] := FALSE;
           #HMI.Selection.Centraggio[1] := FALSE;
       ELSE
           #HMI.Selection.Sollevamento[1] := TRUE;
           #HMI.Selection.Centraggio[1] := TRUE;
       END_IF;

   ELSE
       #Sollevamento[1].Cin.Manager.Rest := TRUE;
       #Centraggio[1].Cin.Manager.Rest := TRUE;
       #HMI.Selection.Sollevamento[1] := FALSE;
       #HMI.Selection.Centraggio[1] := FALSE;

   END_IF;
END_REGION

REGION Network 27: Centraggio - Valve Machine
   RUNG wire#powerrail
      #Centraggio[1](AreaInterface := #AreaInterface, ZSI := #ZSI, DSI := #DSI, DataIn :=, Cin :=, Config := #Config.Centraggio[1], Alarm := #Alarm.Centraggio[1], Warning := #Warning.Centratore[1], MachineInterface =>, COut =>, DataOut =>)
   END_RUNG
   // the same network as SCL:
   #Centraggio[1](AreaInterface := #AreaInterface,   // "ValveMachine_FB"
                  ZSI := #ZSI,
                  DSI := #DSI,
                  Config := #Config.Centraggio[1],
                  Alarm := #Alarm.Centraggio[1],
                  Warning := #Warning.Centratore[1]);
END_REGION

REGION Network 28: Sollevamento - Valve Machine
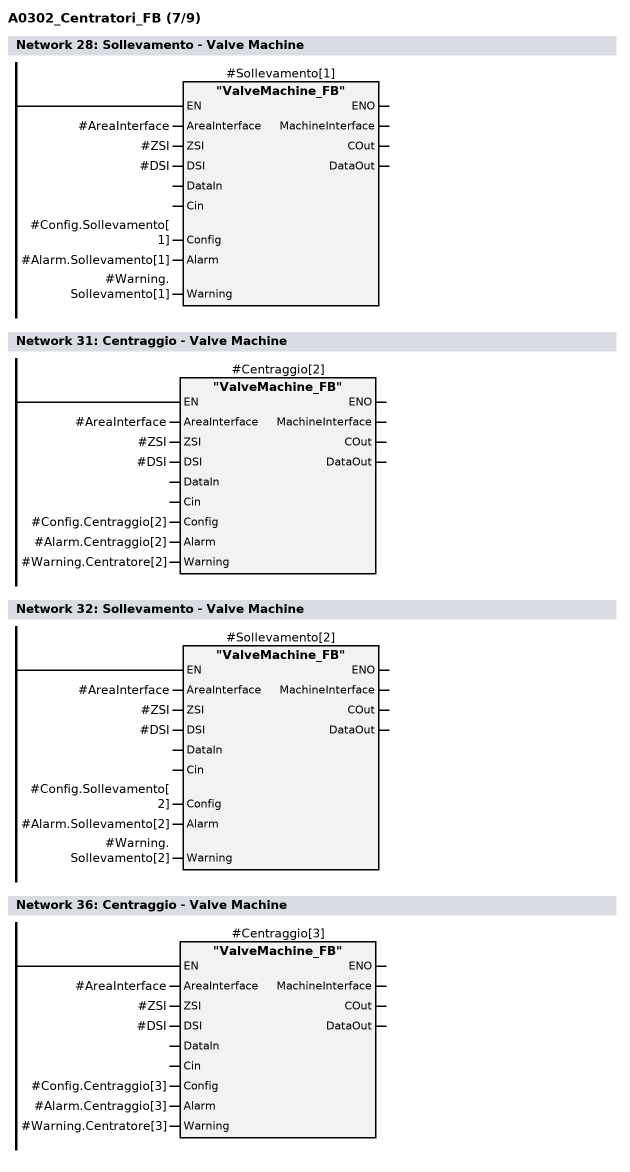
   RUNG wire#powerrail
      #Sollevamento[1](AreaInterface := #AreaInterface, ZSI := #ZSI, DSI := #DSI, DataIn :=, Cin :=, Config := #Config.Sollevamento[1], Alarm := #Alarm.Sollevamento[1], Warning := #Warning.Sollevamento[1], MachineInterface =>, COut =>, DataOut =>)
   END_RUNG
   // the same network as SCL:
   #Sollevamento[1](AreaInterface := #AreaInterface,   // "ValveMachine_FB"
                    ZSI := #ZSI,
                    DSI := #DSI,
                    Config := #Config.Sollevamento[1],
                    Alarm := #Alarm.Sollevamento[1],
                    Warning := #Warning.Sollevamento[1]);
END_REGION

REGION Network 30: <<< CENTRATORE 2 CENTRALE >>>
END_REGION

REGION Network 31: Centraggio - Valve Machine
   RUNG wire#powerrail
      #Centraggio[2](AreaInterface := #AreaInterface, ZSI := #ZSI, DSI := #DSI, DataIn :=, Cin :=, Config := #Config.Centraggio[2], Alarm := #Alarm.Centraggio[2], Warning := #Warning.Centratore[2], MachineInterface =>, COut =>, DataOut =>)
   END_RUNG
   // the same network as SCL:
   #Centraggio[2](AreaInterface := #AreaInterface,   // "ValveMachine_FB"
                  ZSI := #ZSI,
                  DSI := #DSI,
                  Config := #Config.Centraggio[2],
                  Alarm := #Alarm.Centraggio[2],
                  Warning := #Warning.Centratore[2]);
END_REGION

REGION Network 32: Sollevamento - Valve Machine
   RUNG wire#powerrail
      #Sollevamento[2](AreaInterface := #AreaInterface, ZSI := #ZSI, DSI := #DSI, DataIn :=, Cin :=, Config := #Config.Sollevamento[2], Alarm := #Alarm.Sollevamento[2], Warning := #Warning.Sollevamento[2], MachineInterface =>, COut =>, DataOut =>)
   END_RUNG
   // the same network as SCL:
   #Sollevamento[2](AreaInterface := #AreaInterface,   // "ValveMachine_FB"
                    ZSI := #ZSI,
                    DSI := #DSI,
                    Config := #Config.Sollevamento[2],
                    Alarm := #Alarm.Sollevamento[2],
                    Warning := #Warning.Sollevamento[2]);
END_REGION

REGION Network 34: <<< CENTRATORE 3 CODA >>>
END_REGION

REGION Network 35 (SCL): Centraggio - Finestra di lavoro - Enable/Disable
   // Disattivazione Centratore lato Coda in funzione della posizione del Carro Pareggiatore Coda
   // 

   IF #CIn.CarroPareggCoda.Ax.Homed THEN

       IF #CIn.CarroPareggCoda.Ax.ActualPosition >= "PrjConfig_A03".A0302.Centratori.WorkWindows.Coda.Min AND
           #CIn.CarroPareggCoda.Ax.ActualPosition < "PrjConfig_A03".A0302.Centratori.WorkWindows.Coda.Max THEN

           #Sollevamento[3].Cin.Manager.Rest := TRUE;
           #Centraggio[3].Cin.Manager.Rest := TRUE;
           #HMI.Selection.Sollevamento[3] := FALSE;
           #HMI.Selection.Centraggio[3] := FALSE;
       ELSE
           #HMI.Selection.Sollevamento[3] := TRUE;
           #HMI.Selection.Centraggio[3] := TRUE;
       END_IF;

   ELSE
       #Sollevamento[3].Cin.Manager.Rest := TRUE;
       #Centraggio[3].Cin.Manager.Rest := TRUE;
       #HMI.Selection.Sollevamento[3] := FALSE;
       #HMI.Selection.Centraggio[3] := FALSE;

   END_IF;
END_REGION

REGION Network 36: Centraggio - Valve Machine
   RUNG wire#powerrail
      #Centraggio[3](AreaInterface := #AreaInterface, ZSI := #ZSI, DSI := #DSI, DataIn :=, Cin :=, Config := #Config.Centraggio[3], Alarm := #Alarm.Centraggio[3], Warning := #Warning.Centratore[3], MachineInterface =>, COut =>, DataOut =>)
   END_RUNG
   // the same network as SCL:
   #Centraggio[3](AreaInterface := #AreaInterface,   // "ValveMachine_FB"
                  ZSI := #ZSI,
                  DSI := #DSI,
                  Config := #Config.Centraggio[3],
                  Alarm := #Alarm.Centraggio[3],
                  Warning := #Warning.Centratore[3]);
END_REGION

REGION Network 37: Sollevamento - Valve Machine
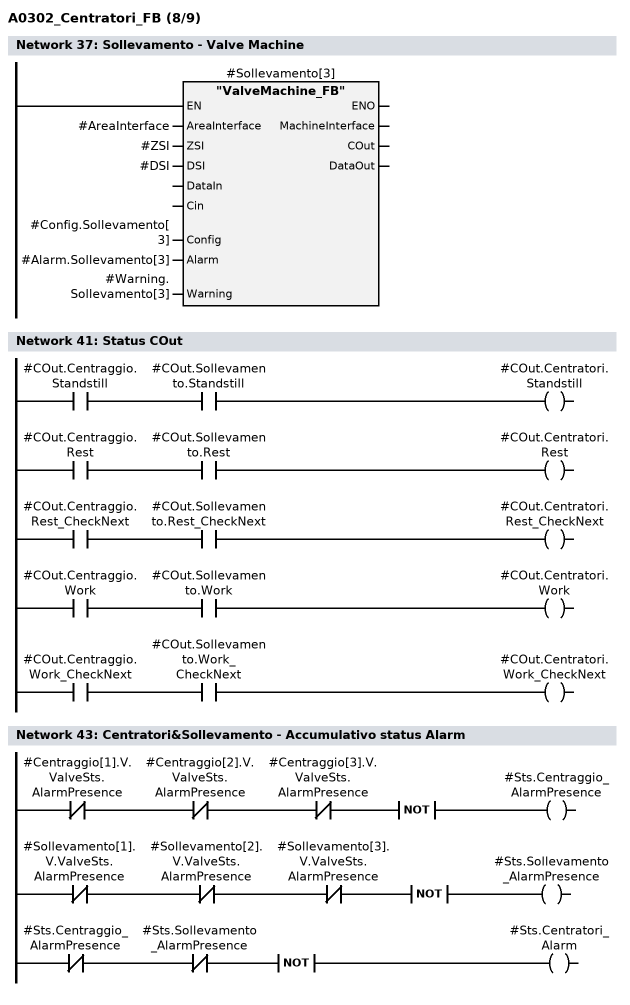
   RUNG wire#powerrail
      #Sollevamento[3](AreaInterface := #AreaInterface, ZSI := #ZSI, DSI := #DSI, DataIn :=, Cin :=, Config := #Config.Sollevamento[3], Alarm := #Alarm.Sollevamento[3], Warning := #Warning.Sollevamento[3], MachineInterface =>, COut =>, DataOut =>)
   END_RUNG
   // the same network as SCL:
   #Sollevamento[3](AreaInterface := #AreaInterface,   // "ValveMachine_FB"
                    ZSI := #ZSI,
                    DSI := #DSI,
                    Config := #Config.Sollevamento[3],
                    Alarm := #Alarm.Sollevamento[3],
                    Warning := #Warning.Sollevamento[3]);
END_REGION

REGION Network 39 (SCL): Centraggio + Sollevamento - COut Centratori
   // Controllo Stato Standstill di tutti i Centraggi
   IF #HMI.Selection.Centraggio[1] AND #HMI.Selection.Centraggio[2] AND #HMI.Selection.Centraggio[3] AND
       #Centraggio[1].Sts.Standstill AND
       #Centraggio[2].Sts.Standstill AND
       #Centraggio[3].Sts.Standstill THEN
       #COut.Centraggio.Standstill := 1;

   ELSIF NOT #HMI.Selection.Centraggio[1] AND #HMI.Selection.Centraggio[2] AND #HMI.Selection.Centraggio[3] AND
       #Centraggio[2].Sts.Standstill AND
       #Centraggio[3].Sts.Standstill THEN
       #COut.Centraggio.Standstill := 1;

   ELSIF #HMI.Selection.Centraggio[1] AND #HMI.Selection.Centraggio[2] AND NOT #HMI.Selection.Centraggio[3] AND
       #Centraggio[1].Sts.Standstill AND
       #Centraggio[2].Sts.Standstill THEN
       #COut.Centraggio.Standstill := 1;

   ELSIF NOT #HMI.Selection.Centraggio[1] AND #HMI.Selection.Centraggio[2] AND NOT #HMI.Selection.Centraggio[3] AND
       #Centraggio[2].Sts.Standstill THEN
       #COut.Centraggio.Standstill := 1;

   ELSE
       #COut.Centraggio.Standstill := 0;
   END_IF;

   // Controllo Stato Standstill di tutti i Sollevamenti

   IF #HMI.Selection.Sollevamento[1] AND #HMI.Selection.Sollevamento[2] AND #HMI.Selection.Sollevamento[3] AND
       #Sollevamento[1].Sts.Standstill AND
       #Sollevamento[2].Sts.Standstill AND
       #Sollevamento[3].Sts.Standstill THEN
       #COut.Sollevamento.Standstill := 1;

   ELSIF NOT #HMI.Selection.Sollevamento[1] AND #HMI.Selection.Sollevamento[2] AND #HMI.Selection.Sollevamento[3] AND
       #Sollevamento[2].Sts.Standstill AND
       #Sollevamento[3].Sts.Standstill THEN
       #COut.Sollevamento.Standstill := 1;

   ELSIF #HMI.Selection.Sollevamento[1] AND #HMI.Selection.Sollevamento[2] AND NOT #HMI.Selection.Sollevamento[3] AND
       #Sollevamento[1].Sts.Standstill AND
       #Sollevamento[2].Sts.Standstill THEN
       #COut.Sollevamento.Standstill := 1;

   ELSIF NOT #HMI.Selection.Sollevamento[1] AND #HMI.Selection.Sollevamento[2] AND NOT #HMI.Selection.Sollevamento[3] AND
       #Sollevamento[2].Sts.Standstill THEN
       #COut.Sollevamento.Standstill := 1;

   ELSE
       #COut.Sollevamento.Standstill := 0;
   END_IF;

   // Controllo uscita COut AT_REST in base allo stato di tutti i Centraggio
   IF #HMI.Selection.Centraggio[1] AND #HMI.Selection.Centraggio[2] AND #HMI.Selection.Centraggio[3] AND
       #Centraggio[1].COut.Rest OR #TON_Anticipi.Rest.Centraggio[1].Q AND
       #Centraggio[2].COut.Rest OR #TON_Anticipi.Rest.Centraggio[2].Q AND
       #Centraggio[3].COut.Rest OR #TON_Anticipi.Rest.Centraggio[3].Q THEN
       #COut.Centraggio.Rest := 1;

   ELSIF NOT #HMI.Selection.Centraggio[1] AND #HMI.Selection.Centraggio[2] AND #HMI.Selection.Centraggio[3] AND
       #Centraggio[2].COut.Rest OR #TON_Anticipi.Rest.Centraggio[2].Q AND
       #Centraggio[3].COut.Rest OR #TON_Anticipi.Rest.Centraggio[3].Q THEN
   #COut.Centraggio.Rest := 1;

   ELSIF #HMI.Selection.Centraggio[1] AND #HMI.Selection.Centraggio[2] AND NOT #HMI.Selection.Centraggio[3] AND
       #Centraggio[1].COut.Rest OR #TON_Anticipi.Rest.Centraggio[1].Q AND
       #Centraggio[2].COut.Rest OR #TON_Anticipi.Rest.Centraggio[2].Q THEN
       #COut.Centraggio.Rest := 1;

   ELSIF NOT #HMI.Selection.Centraggio[1] AND #HMI.Selection.Centraggio[2] AND NOT #HMI.Selection.Centraggio[3] AND
       #Centraggio[2].COut.Rest OR #TON_Anticipi.Rest.Centraggio[2].Q THEN
   #COut.Centraggio.Rest := 1;

   ELSE
   #COut.Centraggio.Rest := 0;
   END_IF;

   // Controllo uscita COut AT_REST in base allo stato di tutti i Sollevamenti
   IF #HMI.Selection.Sollevamento[1] AND #HMI.Selection.Sollevamento[2] AND #HMI.Selection.Sollevamento[3] AND
       #Sollevamento[1].COut.Rest OR #TON_Anticipi.Rest.Sollevamento[1].Q AND
       #Sollevamento[2].COut.Rest OR #TON_Anticipi.Rest.Sollevamento[2].Q AND
       #Sollevamento[3].COut.Rest OR #TON_Anticipi.Rest.Sollevamento[3].Q THEN
       #COut.Sollevamento.Rest := 1;

   ELSIF NOT #HMI.Selection.Sollevamento[1] AND #HMI.Selection.Sollevamento[2] AND #HMI.Selection.Sollevamento[3] AND
       #Sollevamento[2].COut.Rest OR #TON_Anticipi.Rest.Sollevamento[2].Q AND
       #Sollevamento[3].COut.Rest OR #TON_Anticipi.Rest.Sollevamento[3].Q THEN
       #COut.Sollevamento.Rest := 1;

   ELSIF #HMI.Selection.Sollevamento[1] AND #HMI.Selection.Sollevamento[2] AND NOT #HMI.Selection.Sollevamento[3] AND
       #Sollevamento[1].COut.Rest OR #TON_Anticipi.Rest.Sollevamento[1].Q AND
       #Sollevamento[2].COut.Rest OR #TON_Anticipi.Rest.Sollevamento[2].Q THEN
       #COut.Sollevamento.Rest := 1;

   ELSIF NOT #HMI.Selection.Sollevamento[1] AND #HMI.Selection.Sollevamento[2] AND NOT #HMI.Selection.Sollevamento[3] AND
       #Sollevamento[2].COut.Rest OR #TON_Anticipi.Rest.Sollevamento[2].Q THEN
       #COut.Sollevamento.Rest := 1;

   ELSE
       #COut.Sollevamento.Rest := 0;
   END_IF;

   // Controllo uscita COut AT_WORK in base allo stato di tutti i Centraggio
   IF #HMI.Selection.Centraggio[1] AND #HMI.Selection.Centraggio[2] AND #HMI.Selection.Centraggio[3] AND
       #Centraggio[1].COut.Work OR #TON_Anticipi.Rest.Centraggio[1].Q AND
       #Centraggio[2].COut.Work OR #TON_Anticipi.Rest.Centraggio[2].Q AND
       #Centraggio[3].COut.Work OR #TON_Anticipi.Rest.Centraggio[3].Q THEN
       #COut.Centraggio.Work := 1;

   ELSIF NOT #HMI.Selection.Centraggio[1] AND #HMI.Selection.Centraggio[2] AND #HMI.Selection.Centraggio[3] AND
       #Centraggio[2].COut.Work OR #TON_Anticipi.Rest.Centraggio[2].Q AND
       #Centraggio[3].COut.Work OR #TON_Anticipi.Rest.Centraggio[3].Q THEN
       #COut.Centraggio.Work := 1;

   ELSIF #HMI.Selection.Centraggio[1] AND #HMI.Selection.Centraggio[2] AND NOT #HMI.Selection.Centraggio[3] AND
       #Centraggio[1].COut.Work OR #TON_Anticipi.Rest.Centraggio[1].Q AND
       #Centraggio[2].COut.Work OR #TON_Anticipi.Rest.Centraggio[2].Q THEN
       #COut.Centraggio.Work := 1;

   ELSIF NOT #HMI.Selection.Centraggio[1] AND #HMI.Selection.Centraggio[2] AND NOT #HMI.Selection.Centraggio[3] AND
       #Centraggio[2].COut.Work OR #TON_Anticipi.Rest.Centraggio[2].Q THEN
       #COut.Centraggio.Work := 1;

   ELSE
       #COut.Centraggio.Work := 0;
   END_IF;

   // Controllo uscita COut AT_WORK in base allo stato di tutti i Sollevamenti
   IF #HMI.Selection.Sollevamento[1] AND #HMI.Selection.Sollevamento[2] AND #HMI.Selection.Sollevamento[3] AND
       #Sollevamento[1].COut.Work OR #TON_Anticipi.Work.Sollevamento[1].Q AND
       #Sollevamento[2].COut.Work OR #TON_Anticipi.Work.Sollevamento[2].Q AND
       #Sollevamento[3].COut.Work OR #TON_Anticipi.Work.Sollevamento[3].Q THEN
       #COut.Sollevamento.Work := 1;

   ELSIF NOT #HMI.Selection.Sollevamento[1] AND #HMI.Selection.Sollevamento[2] AND #HMI.Selection.Sollevamento[3] AND
       #Sollevamento[2].COut.Work OR #TON_Anticipi.Work.Sollevamento[2].Q AND
       #Sollevamento[3].COut.Work OR #TON_Anticipi.Work.Sollevamento[3].Q THEN
       #COut.Sollevamento.Work := 1;

   ELSIF #HMI.Selection.Sollevamento[1] AND #HMI.Selection.Sollevamento[2] AND NOT #HMI.Selection.Sollevamento[3] AND
       #Sollevamento[1].COut.Work OR #TON_Anticipi.Work.Sollevamento[1].Q AND
       #Sollevamento[2].COut.Work OR #TON_Anticipi.Work.Sollevamento[2].Q THEN
       #COut.Sollevamento.Work := 1;

   ELSIF NOT #HMI.Selection.Sollevamento[1] AND #HMI.Selection.Sollevamento[2] AND NOT #HMI.Selection.Sollevamento[3] AND
       #Sollevamento[2].COut.Work OR #TON_Anticipi.Work.Sollevamento[2].Q THEN
       #COut.Sollevamento.Work := 1;

   ELSE
       #COut.Sollevamento.Work := 0;
   END_IF;
END_REGION

REGION Network 41: Status COut
   RUNG wire#powerrail
      Contact( #COut.Centraggio.Standstill )
      Contact( #COut.Sollevamento.Standstill )
      Coil( #COut.Centratori.Standstill )
   END_RUNG
   RUNG wire#powerrail
      Contact( #COut.Centraggio.Rest )
      Contact( #COut.Sollevamento.Rest )
      Coil( #COut.Centratori.Rest )
   END_RUNG
   RUNG wire#powerrail
      Contact( #COut.Centraggio.Rest_CheckNext )
      Contact( #COut.Sollevamento.Rest_CheckNext )
      Coil( #COut.Centratori.Rest_CheckNext )
   END_RUNG
   RUNG wire#powerrail
      Contact( #COut.Centraggio.Work )
      Contact( #COut.Sollevamento.Work )
      Coil( #COut.Centratori.Work )
   END_RUNG
   RUNG wire#powerrail
      Contact( #COut.Centraggio.Work_CheckNext )
      Contact( #COut.Sollevamento.Work_CheckNext )
      Coil( #COut.Centratori.Work_CheckNext )
   END_RUNG
   // the same network as SCL:
   #COut.Centratori.Standstill := #COut.Centraggio.Standstill AND #COut.Sollevamento.Standstill;
   #COut.Centratori.Rest := #COut.Centraggio.Rest AND #COut.Sollevamento.Rest;
   #COut.Centratori.Rest_CheckNext := #COut.Centraggio.Rest_CheckNext AND #COut.Sollevamento.Rest_CheckNext;
   #COut.Centratori.Work := #COut.Centraggio.Work AND #COut.Sollevamento.Work;
   #COut.Centratori.Work_CheckNext := #COut.Centraggio.Work_CheckNext AND #COut.Sollevamento.Work_CheckNext;
END_REGION

REGION Network 43: Centratori&Sollevamento - Accumulativo status Alarm
   RUNG wire#powerrail
      I_Contact( #Centraggio[1].V.ValveSts.AlarmPresence )
      I_Contact( #Centraggio[2].V.ValveSts.AlarmPresence )
      I_Contact( #Centraggio[3].V.ValveSts.AlarmPresence )
      Not()
      Coil( #Sts.Centraggio_AlarmPresence )
   END_RUNG
   RUNG wire#powerrail
      I_Contact( #Sollevamento[1].V.ValveSts.AlarmPresence )
      I_Contact( #Sollevamento[2].V.ValveSts.AlarmPresence )
      I_Contact( #Sollevamento[3].V.ValveSts.AlarmPresence )
      Not()
      Coil( #Sts.Sollevamento_AlarmPresence )
   END_RUNG
   RUNG wire#powerrail
      I_Contact( #Sts.Centraggio_AlarmPresence )
      I_Contact( #Sts.Sollevamento_AlarmPresence )
      Not()
      Coil( #Sts.Centratori_Alarm )
   END_RUNG
   // the same network as SCL:
   #Sts.Centraggio_AlarmPresence := NOT (NOT #Centraggio[1].V.ValveSts.AlarmPresence AND NOT #Centraggio[2].V.ValveSts.AlarmPresence AND NOT #Centraggio[3].V.ValveSts.AlarmPresence);
   #Sts.Sollevamento_AlarmPresence := NOT (NOT #Sollevamento[1].V.ValveSts.AlarmPresence AND NOT #Sollevamento[2].V.ValveSts.AlarmPresence AND NOT #Sollevamento[3].V.ValveSts.AlarmPresence);
   #Sts.Centratori_Alarm := NOT (NOT #Sts.Centraggio_AlarmPresence AND NOT #Sts.Sollevamento_AlarmPresence);
END_REGION

REGION Network 44 (SCL): HMI STATUS - Postazione
   // Area dati appoggio per HMI
   // CENTRATORI
   #HMI.Centraggio_Sts.Standstill := #COut.Centraggio.Standstill;
   #HMI.Centraggio_Sts.Rest := #COut.Centraggio.Rest;
   #HMI.Centraggio_Sts.Work := #COut.Centraggio.Work;
   #HMI.Centraggio_Sts.AlarmPresence := #Sts.Centraggio_AlarmPresence;

   // SOLLEVAMENTO
   #HMI.Sollevamento_Sts.Standstill := #COut.Sollevamento.Standstill;
   #HMI.Sollevamento_Sts.Rest := #COut.Sollevamento.Rest;
   #HMI.Sollevamento_Sts.Work := #COut.Sollevamento.Work;
   #HMI.Sollevamento_Sts.AlarmPresence := #Sts.Sollevamento_AlarmPresence;

   // STAZIONE CENTRATORI
   #HMI.Centratori_Sts.Standstill := #COut.Centratori.Standstill;
   #HMI.Centratori_Sts.Rest := #COut.Centratori.Rest;
   #HMI.Centratori_Sts.Work := #COut.Centratori.Work;
   #HMI.Centratori_Sts.AlarmPresence := #Sts.Centratori_Alarm;
END_REGION

REGION Network 45: <<< MACHINE STATUS >>>
END_REGION

REGION Network 46: Collect machine to zone interface (internal machines OR)
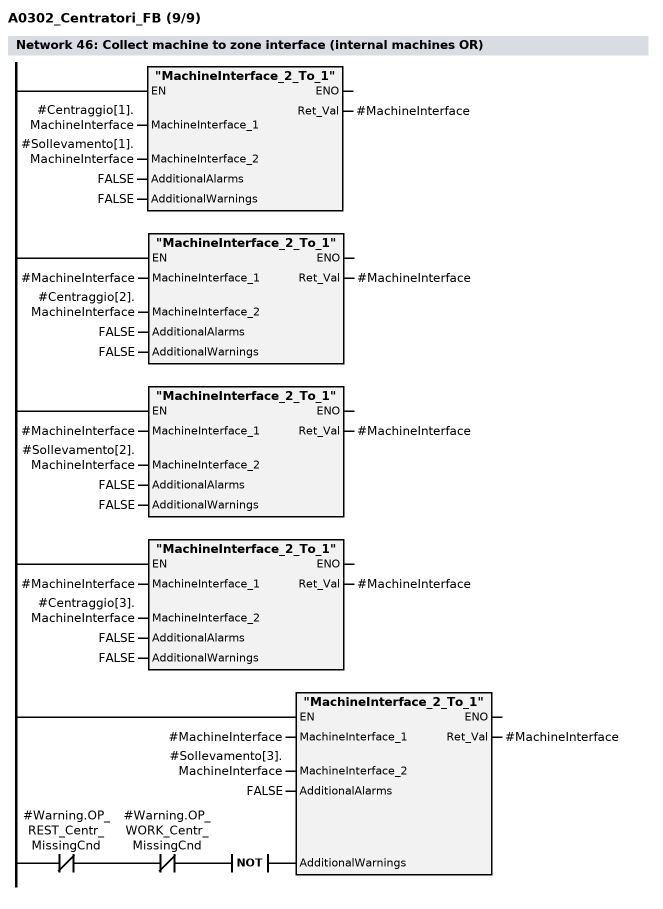
   RUNG wire#powerrail
      "MachineInterface_2_To_1"(MachineInterface_1 := #Centraggio[1].MachineInterface, MachineInterface_2 := #Sollevamento[1].MachineInterface, AdditionalAlarms := FALSE, AdditionalWarnings := FALSE, Ret_Val => #MachineInterface)
   END_RUNG
   RUNG wire#powerrail
      "MachineInterface_2_To_1"(MachineInterface_1 := #MachineInterface, MachineInterface_2 := #Centraggio[2].MachineInterface, AdditionalAlarms := FALSE, AdditionalWarnings := FALSE, Ret_Val => #MachineInterface)
   END_RUNG
   RUNG wire#powerrail
      "MachineInterface_2_To_1"(MachineInterface_1 := #MachineInterface, MachineInterface_2 := #Sollevamento[2].MachineInterface, AdditionalAlarms := FALSE, AdditionalWarnings := FALSE, Ret_Val => #MachineInterface)
   END_RUNG
   RUNG wire#powerrail
      "MachineInterface_2_To_1"(MachineInterface_1 := #MachineInterface, MachineInterface_2 := #Centraggio[3].MachineInterface, AdditionalAlarms := FALSE, AdditionalWarnings := FALSE, Ret_Val => #MachineInterface)
   END_RUNG
   RUNG wire#powerrail
      "MachineInterface_2_To_1"(AdditionalWarnings := wire#w1, MachineInterface_1 := #MachineInterface, MachineInterface_2 := #Sollevamento[3].MachineInterface, AdditionalAlarms := FALSE, Ret_Val => #MachineInterface)
   END_RUNG
   RUNG wire#powerrail
      I_Contact( #Warning.OP_REST_Centr_MissingCnd )
      I_Contact( #Warning.OP_WORK_Centr_MissingCnd )
      Not()
   END_RUNG wire#w1
   // the same network as SCL:
   #MachineInterface := "MachineInterface_2_To_1"(MachineInterface_1 := #Centraggio[1].MachineInterface,
                           MachineInterface_2 := #Sollevamento[1].MachineInterface,
                           AdditionalAlarms := FALSE,
                           AdditionalWarnings := FALSE);
   #MachineInterface := "MachineInterface_2_To_1"(MachineInterface_1 := #MachineInterface,
                           MachineInterface_2 := #Centraggio[2].MachineInterface,
                           AdditionalAlarms := FALSE,
                           AdditionalWarnings := FALSE);
   #MachineInterface := "MachineInterface_2_To_1"(MachineInterface_1 := #MachineInterface,
                           MachineInterface_2 := #Sollevamento[2].MachineInterface,
                           AdditionalAlarms := FALSE,
                           AdditionalWarnings := FALSE);
   #MachineInterface := "MachineInterface_2_To_1"(MachineInterface_1 := #MachineInterface,
                           MachineInterface_2 := #Centraggio[3].MachineInterface,
                           AdditionalAlarms := FALSE,
                           AdditionalWarnings := FALSE);
   #MachineInterface := "MachineInterface_2_To_1"(MachineInterface_1 := #MachineInterface,
                           MachineInterface_2 := #Sollevamento[3].MachineInterface,
                           AdditionalAlarms := FALSE,
                           AdditionalWarnings := NOT (NOT #Warning.OP_REST_Centr_MissingCnd AND NOT #Warning.OP_WORK_Centr_MissingCnd));
END_REGION
END_FUNCTION_BLOCK
